// TIA Portal V18 export
FUNCTION_BLOCK "LoadCell"   // FB7, LAD
TITLE = Description:
{ S7_Optimized_Access := 'TRUE' }
VERSION : 0.1
// Old control block - should be checked described.
// stored: AutoNumber true, IsIECCheckEnabled false, IsRetainMemResEnabled false, MemoryReserve 100, SetENOAutomatically false, UDAEnableTagReadback false
   VAR_INPUT
      MinValue : UInt := 0;
      MaxValue : UInt := 27648;
      ILoadCell : UInt;
      Const_V : UInt := 10;
      Const_SubWeight : Real := 0.629;
      Const_Kg : UInt := 13970;
   END_VAR
   VAR_OUTPUT
      OWeight : UInt;
   END_VAR
   VAR_TEMP
      NormVal : Real;
      ScalVal : Real;
      SubVal : Real;
      MulVal : Real;
   END_VAR
BEGIN

REGION Network 1
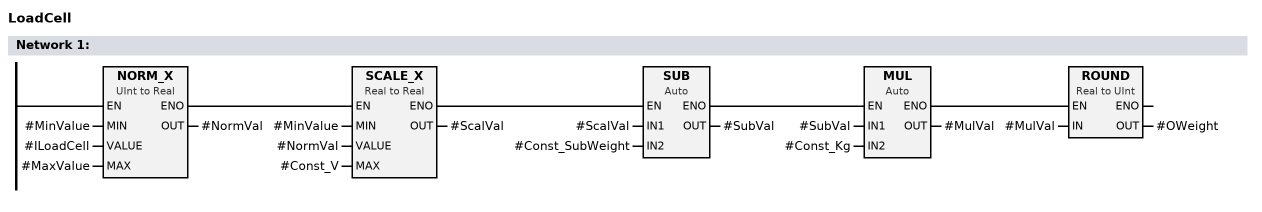
   RUNG wire#powerrail
      { S7_Templates := "[SrcType := UInt, DestType := Real]" } Normalize(min := #MinValue, value := #ILoadCell, max := #MaxValue, out => #NormVal)
      { S7_Templates := "[SrcType := Real, DestType := Real]" } Scale(min := #MinValue, value := #NormVal, max := #Const_V, out => #ScalVal)
      Sub(in1 := #ScalVal, in2 := #Const_SubWeight, out => #SubVal)
      Mul(in1 := #SubVal, in2 := #Const_Kg, out => #MulVal)
      { S7_Templates := "[SrcType := Real, DestType := UInt]" } Round(in := #MulVal, out => #OWeight)
   END_RUNG
   // the same network as SCL:
   #NormVal := NORM_X(MIN := #MinValue, VALUE := #ILoadCell, MAX := #MaxValue);
   #ScalVal := SCALE_X(MIN := #MinValue, VALUE := #NormVal, MAX := #Const_V);
   #SubVal := #ScalVal - #Const_SubWeight;
   #MulVal := #SubVal * #Const_Kg;
   #OWeight := ROUND(#MulVal);
END_REGION
END_FUNCTION_BLOCK
